FUNCTION ArrayBool_TO_ArrayByte 
VAR_INPUT
	In:					POINTER TO BOOL;// Bool数组
	InLen:				INT;// sizeof(In)
	Out:				POINTER TO BYTE;// Byte数组
	OutLen:				INT;// sizeof(Out)
END_VAR
VAR
	i:					INT;
	t:					INT;
	temp:				ARRAY[0..7] OF BOOL;
	inCount:			INT;
END_VAR

IF InLen<>OutLen*8 THEN
	RETURN;
END_IF

FOR i:=0 TO OutLen-1 BY 1 DO
	FOR t:=0 TO 7 BY 1 DO
		temp[t]:=In[inCount];
		inCount:=inCount+1;
	END_FOR
	Out[i]:=ArrayBool_TO_Byte(ADR(temp),SIZEOF(temp));
END_FOR

END_FUNCTION

(* stored: Version 1.1.0.1, ProductVersion 3.1.4024.3
   POU ArrayBool_TO_ArrayByte: Id {997e0eeb-eefd-485a-959b-e5f5b0f4f731}, SpecialFunc None *)
